PROGRAM MAIN
VAR
END_VAR

// Generating some new stuff to test Git

END_PROGRAM

(* stored: Version 1.1.0.1, ProductVersion 3.1.4024.12
   POU MAIN: Id {aa9c1110-05c8-4a57-8d0e-3ce20f961eb8}, SpecialFunc None *)
